//Search Startup values for enter the room
	fbSearchStartUpLevel 		: FB_SearchStartUpLevel_EX ;
	
END_VAR

VAR_IN_OUT
	stTuneData					: ST_TuneData_EX;
	stPirSensorData				: ST_DALI_Sensor;
	stLiveData					: ST_LiveData;
END_VAR

fbBallast(nCycleTimeInMS := nCycleTimeInMS);


A_TuningProcess();
A_RoomFct();

A_DaliUpdate();

ACTION A_DaliUpdate:

	IF stDaliSetup.DALI_LINE_NUM_PRIM <> 0 THEN
		
		stLgtCmd_Prim.bSetCtrlValDct:= fbLightCtrl_2Rows.bWriteValue ;
		stLgtCmd_Prim.fSetCtrlValDct:= fbLightCtrl_2Rows.fSP_Room;
		stLgtCmd_Prim.bDimDwn := fbLightCtrl_2Rows.bDimDwn;
		stLgtCmd_Prim.bDimUp := fbLightCtrl_2Rows.bDimUp;
		
		stLgtCmd_Prim.bClMinCtrlVal:= fbLightCtrl_2Rows.bClMinCtrlVal;
		
		fbBallast.M_PrimBallast(
				byShrtAdr_Prim:= stDaliSetup.byShrtAdr_Prim, 
				byGrpAdr_Prim:= stDaliSetup.byGrpAdr_Prim, 
				eMod_Prim:= stDaliSetup.eMod_Prim, 
				stLgtCmd_Prim:= stLgtCmd_Prim, 
				DALI_LINE_NUM:=stDaliSetup.DALI_LINE_NUM_PRIM,
				bUseGlobalFadeTimeSettings:= stDaliSetup.bLocal_GlobalFadeInfo , 
				bReInit:= bReInit, 
				bTurnOff:=fbLightCtrl.bOffZone1 , 
				ipCommunication:= ipCommunication_Prim );
	END_IF 
	
	IF stDaliSetup.DALI_LINE_NUM_SEC <> 0 THEN

		stLgtCmd_Sec.bSetCtrlValDct:= fbLightCtrl_2Rows.bWriteValue ;
		stLgtCmd_Sec.fSetCtrlValDct:=fbLightCtrl_2Rows.fSP_Window;
		stLgtCmd_Sec.bDimDwn := fbLightCtrl_2Rows.bDimDwn;
		stLgtCmd_Sec.bDimUp := fbLightCtrl_2Rows.bDimUp;		

		stLgtCmd_Sec.bClMinCtrlVal:= fbLightCtrl_2Rows.bClMinCtrlVal;
	
		fbBallast.M_SecBallast(
			byShrtAdr_Sec:= stDaliSetup.byShrtAdr_Sec, 
			byGrpAdr_Sec:= stDaliSetup.byGrpAdr_Sec, 
			eMod_Sec:= stDaliSetup.eMod_Sec, 
			stLgtCmd_Sec:= stLgtCmd_Sec, 
			DALI_LINE_NUM:=stDaliSetup.DALI_LINE_NUM_SEC,
			bUseGlobalFadeTimeSettings:= stDaliSetup.bLocal_GlobalFadeInfo , 
			bReInit:= bReInit, 
			bTurnOff:=fbLightCtrl.bOffZone2 , 
			ipCommunication:= ipCommunication_Sec );		
	END_IF 
	
	IF stDaliSetup.DALI_LINE_NUM_SUPL <> 0 THEN
	
		fbBallast.M_SuplBallast(
			byShrtAdr_Supl:= stDaliSetup.byShrtAdr_Supl, 
			byGrpAdr_Supl:= stDaliSetup.byGrpAdr_Supl, 
			eMod_Supl:= stDaliSetup.eMod_Supl, 
			stLgtCmd_Supl:= stLgtCmd_Supl, 
			DALI_LINE_NUM:=stDaliSetup.DALI_LINE_NUM_SUPL,
			bUseGlobalFadeTimeSettings:= stDaliSetup.bLocal_GlobalFadeInfo , 
			bReInit:= bReInit, 
			bTurnOff:= fbLightCtrl.bOffZone2 , 
			ipCommunication:= ipCommunication_Supl );
	END_IF
END_ACTION

ACTION A_RoomFct:

fbLightCtrl(
	bTopButtonZone1:= bButtonZone1,
	bBottomButtonZone1 := bBottomButtonZone1,
	bButtonZone2:= bButtonZone2,
	bTopButtonOverride:= bTopButtonOverride,
	bBottomButtonOverride:= bBottomButtonOverride,
	bNoButtons:= bNoButtons,
	bPIR:= stPirSensorData.bPrc, 
	fLuxOn:= fLuxOn, 
	fLuxDim:= fLuxDim, 
	tPIRDim:= tPIRDim, 
	tPIROff:= tPIROff, 
	fLuxZone1=> , 
	bDimUp=> , 
	bDimDwn=> , 
	bOnZone1=> bOccupiedRoom, 
	bOffZone1=> , 
	bAutoZone2=> , 
	bOnZone2=> , 
	bOffZone2=> );

bEnableLightCtrl:= fbLightCtrl.bOnZone1 AND fbLightCtrl.bAutoZone1;

fbRTrigStartCtrl(CLK:= fbAutoTuneStartUpLevels.bTuningDone AND bEnableLightCtrl);
fbStartStopLightCtrl(SET1 :=fbRTrigStartCtrl.Q , RESET:= NOT bEnableLightCtrl OR fbLightCtrl.bDimDwn OR fbLightCtrl.bDimUp );

fbSearchStartUpLevel(
	bSearch:= fbStartStopLightCtrl.Q1, 
	fSp:= fbLightCtrl.fLuxZone1, 
	stPirSensorData:= stPirSensorData, 
	bSync=> , 
	fSttUpCtrlVal=> , 
	stTuneData:=stTuneData );
	
fbLightCtrl_2Rows(
	_bEnable:=  fbStartStopLightCtrl.Q1, 
	_bSyncVal:=fbSearchStartUpLevel.bSync , 
	_fSyncVal:= fbSearchStartUpLevel.fSttUpCtrlVal, 
	_fSP:= fbLightCtrl.fLuxZone1, 
	_fPV:=stPirSensorData.fBrightness , 
	_fStep1Limit:= 8, 
	_fSPStep1:= 0.5, 
	_fStep2Limit:= 16, 
	_fSPStep2:= 1, 
	_fStep3Limit:= 24, 
	_fSPStep3:= 1.5, 
	_fStep4Limit:= 34, 
	_fSPStep4:= 2.0, 
	_fStep5Limit:= 40, 
	_fSPStep5:= 2.5, 
	_tStepTime:= T#10S, 																											//Testing 10s (originally 15s)
	_bStepModeCalculationOnSP:= FALSE , 
	_bTuningInProcess:= bTunningInProcess, 
	_bSetValDct:= fbAutoTuneStartUpLevels.bSetValDct, 
	_fSetValDct:= fbAutoTuneStartUpLevels.fSetValDct, 
	_bDimUp:= fbLightCtrl.bDimUp, 
	_bDimDown:= fbLightCtrl.bDimDwn, 
	_bOff:= fbLightCtrl.bOffZone1, 
	_fRowOffset:= fOffsetSec, 
	_fActlLgtLvl_Prim:= fbBallast.fActlLgtLvl_Prim, 
	_fActlLgtLvl_Sec:= fbBallast.fActlLgtLvl_Sec, 
	_bRecallManualLevel:= , 
	_fMinOutputPowerLevel := fMinOutputPowerLevelRoom ,
	_fMaxOutputPowerLevel := fMaxOutputPowerLevelRoom,
	_DALI_LINE_NUM_SEC	:= stDaliSetup.DALI_LINE_NUM_SEC,
	fSP_Window=> , 
	fSP_Room=> , 
	bWriteValue=> , 
	bDimUp=> , 
	bDimDwn=> , 
	bOff=> , 
	bClMinCtrlVal=> ,
	stPirSensorData:=stPirSensorData);
	
//Supplement light
fbLightCtrl_Supl(
	bSwi:= , 
	bSwiUp:= , 
	bSwiDwn:= , 
	udiSwiOvrTi:= , 
	bUp:= , 
	bDwn:= , 
	bOn:=fbLightCtrl.bOnZone2 , 
	bOff:= fbLightCtrl.bOffZone2, 
	eOnMod:= , 
	fOnVal:= , 
	bClMinVal:= , 
	bClMaxVal:= , 
	bSetValDct:= , 
	fSetValDct:= , 
	fActlLgtLvl:= fbBallast.fActlLgtLvl_Supl, 
	stLgtCmd=> stLgtCmd_Supl);
END_ACTION

ACTION A_TuningProcess:

fbAutoTuneStartUpLevels(
	bRunTuning:= (NOT stTuneData.bTunnigDone AND stPirSensorData.fBrightness < 25) OR bRunTuning, 
	tTuningDelay:= DALI_Param.tOutTuneDelay, 
	bTuningInProcess=> bTunningInProcess, 
	sActProcess=> , 
	bTuningDone=> , 
	bSetValDct=> , 
	fSetValDct=> , 
	stTuneData:=stTuneData,
 	stPirSensorData:= stPirSensorData);
END_ACTION

END_FUNCTION_BLOCK

// POUs/Templates/FB_Light_Type_B
FUNCTION_BLOCK FB_Light_Type_B
VAR_INPUT	
	nZoneID						: UDINT;
	bButtonZone1				: BOOL;
	bBottomButtonZone1			: BOOL;
	bButtonZone2				: BOOL;
	bTopButtonOverride		: BOOL;
	bBottomButtonOverride	: BOOL;
	bNoButtons					: BOOL;
	bNeighborRoomsPir			: BOOL;
	fLuxOn 						: REAL;
	fLuxDim						: REAL;
	tPIRDim						: TIME;
	tPIROff						: TIME;
	fOffsetSec					: REAL;
	bReInit						: BOOL;
	stDaliSetup					: ST_DALI_RoomSetup;
	ipCommunication_Prim		: I_DALICommunication;
	ipCommunication_Sec			: I_DALICommunication;
	ipCommunication_Supl		: I_DALICommunication;
	fMinOutputPowerLevelRoom 	: REAL;
	fMaxOutputPowerLevelRoom	: REAL;
	nCycleTimeInMS				: UDINT;
	bRunTuning 					: BOOL;
END_VAR
VAR_OUTPUT
	bOccupiedRoom 	: BOOL;
	bError_Prim 	: BOOL;
	nError_Prim 	: UINT;
END_VAR
VAR
	fbBallast					: FB_Light_Ballast;
	fbLightCtrl					: FB_FunctionType_A ;
	fbShortLongPresZone1 		: FB_Click;
	fbShortLongPressBottomZone1 : FB_Click;
	fbShortLongPresZone2 		: FB_Click;

	stLgtCmd_Prim				: ST_LgtCmd;
	stLgtCmd_Sec				: ST_LgtCmd;
	stLgtCmd_Supl				: ST_LgtCmd;
	
	fbLightCtrl_2Rows			: FB_LightCtrl_2Groups;
	fbLightCtrl_Supl			: FB_LightSwitch;

	bTunningInProcess			: BOOL;
	bEnableLightCtrl			: BOOL;
	fbRTrigStartCtrl 			: R_TRIG;
	
	bAnyPir						: BOOL;

//Tuning data
	fbPulsReadSensorData_TON	: TON;
	fbAutoTuneStartUpLevels		: FB_AutoTune_TcBA_Ex;
	fbR_TrigTuningDone			: R_TRIG ;
	fbStartStopLightCtrl: SR;
	
//Search Startup values for enter the room
	fbSearchStartUpLevel 		: FB_SearchStartUpLevel_EX ;
	
END_VAR

VAR_IN_OUT
	stTuneData					: ST_TuneData_EX;
	stPirSensorData				: ST_DALI_Sensor;
	stLiveData					: ST_LiveData;
END_VAR

fbBallast(nCycleTimeInMS := nCycleTimeInMS);


A_TuningProcess();
A_RoomFct();

A_DaliUpdate();

ACTION A_DaliUpdate:

	IF stDaliSetup.DALI_LINE_NUM_PRIM <> 0 THEN
		
		stLgtCmd_Prim.bSetCtrlValDct:= fbLightCtrl_2Rows.bWriteValue ;
		stLgtCmd_Prim.fSetCtrlValDct:= fbLightCtrl_2Rows.fSP_Room;
		stLgtCmd_Prim.bDimDwn := fbLightCtrl_2Rows.bDimDwn;
		stLgtCmd_Prim.bDimUp := fbLightCtrl_2Rows.bDimUp;
		
		stLgtCmd_Prim.bClMinCtrlVal:= fbLightCtrl_2Rows.bClMinCtrlVal;
		
		fbBallast.M_PrimBallast(
				byShrtAdr_Prim:= stDaliSetup.byShrtAdr_Prim, 
				byGrpAdr_Prim:= stDaliSetup.byGrpAdr_Prim, 
				eMod_Prim:= stDaliSetup.eMod_Prim, 
				stLgtCmd_Prim:= stLgtCmd_Prim, 
				DALI_LINE_NUM:=stDaliSetup.DALI_LINE_NUM_PRIM,
				bUseGlobalFadeTimeSettings:= stDaliSetup.bLocal_GlobalFadeInfo , 
				bReInit:= bReInit, 
				bTurnOff:=fbLightCtrl.bOffZone1 , 
				ipCommunication:= ipCommunication_Prim );
	END_IF 
	
	IF stDaliSetup.DALI_LINE_NUM_SEC <> 0 THEN

		stLgtCmd_Sec.bSetCtrlValDct:= fbLightCtrl_2Rows.bWriteValue ;
		stLgtCmd_Sec.fSetCtrlValDct:=fbLightCtrl_2Rows.fSP_Window;
		stLgtCmd_Sec.bDimDwn := fbLightCtrl_2Rows.bDimDwn;
		stLgtCmd_Sec.bDimUp := fbLightCtrl_2Rows.bDimUp;		

		stLgtCmd_Sec.bClMinCtrlVal:= fbLightCtrl_2Rows.bClMinCtrlVal;
	
		fbBallast.M_SecBallast(
			byShrtAdr_Sec:= stDaliSetup.byShrtAdr_Sec, 
			byGrpAdr_Sec:= stDaliSetup.byGrpAdr_Sec, 
			eMod_Sec:= stDaliSetup.eMod_Sec, 
			stLgtCmd_Sec:= stLgtCmd_Sec, 
			DALI_LINE_NUM:=stDaliSetup.DALI_LINE_NUM_SEC,
			bUseGlobalFadeTimeSettings:= stDaliSetup.bLocal_GlobalFadeInfo , 
			bReInit:= bReInit, 
			bTurnOff:=fbLightCtrl.bOffZone2 , 
			ipCommunication:= ipCommunication_Sec );		
	END_IF 
	
	IF stDaliSetup.DALI_LINE_NUM_SUPL <> 0 THEN
	
		fbBallast.M_SuplBallast(
			byShrtAdr_Supl:= stDaliSetup.byShrtAdr_Supl, 
			byGrpAdr_Supl:= stDaliSetup.byGrpAdr_Supl, 
			eMod_Supl:= stDaliSetup.eMod_Supl, 
			stLgtCmd_Supl:= stLgtCmd_Supl, 
			DALI_LINE_NUM:=stDaliSetup.DALI_LINE_NUM_SUPL,
			bUseGlobalFadeTimeSettings:= stDaliSetup.bLocal_GlobalFadeInfo , 
			bReInit:= bReInit, 
			bTurnOff:= fbLightCtrl.bOffZone2 , 
			ipCommunication:= ipCommunication_Supl );
	END_IF
END_ACTION

ACTION A_RoomFct:
bAnyPir	:= stPirSensorData.bPrc OR bNeighborRoomsPir;

fbLightCtrl(
	bTopButtonZone1:= bButtonZone1,
	bBottomButtonZone1 := bBottomButtonZone1,
	bButtonZone2:= bButtonZone2,
	bTopButtonOverride:= bTopButtonOverride,
	bBottomButtonOverride:= bBottomButtonOverride,
	bNoButtons:= bNoButtons,
	bPIR:= bAnyPir, 
	fLuxOn:= fLuxOn, 
	fLuxDim:= fLuxDim, 
	tPIRDim:= tPIRDim, 
	tPIROff:= tPIROff, 
	fLuxZone1=> , 
	bDimUp=> , 
	bDimDwn=> , 
	bOnZone1=> bOccupiedRoom, 
	bOffZone1=> , 
	bAutoZone2=> , 
	bOnZone2=> , 
	bOffZone2=> );

bEnableLightCtrl:= fbLightCtrl.bOnZone1 AND fbLightCtrl.bAutoZone1;

fbRTrigStartCtrl(CLK:= fbAutoTuneStartUpLevels.bTuningDone AND bEnableLightCtrl);
fbStartStopLightCtrl(SET1 :=fbRTrigStartCtrl.Q , RESET:= NOT bEnableLightCtrl OR fbLightCtrl.bDimDwn OR fbLightCtrl.bDimUp );

fbSearchStartUpLevel(
	bSearch:= fbStartStopLightCtrl.Q1, 
	fSp:= fbLightCtrl.fLuxZone1, 
	stPirSensorData:= stPirSensorData, 
	bSync=> , 
	fSttUpCtrlVal=> , 
	stTuneData:=stTuneData );
	
fbLightCtrl_2Rows(
	_bEnable:=  fbStartStopLightCtrl.Q1, 
	_bSyncVal:=fbSearchStartUpLevel.bSync , 
	_fSyncVal:= fbSearchStartUpLevel.fSttUpCtrlVal, 
	_fSP:= fbLightCtrl.fLuxZone1, 
	_fPV:=stPirSensorData.fBrightness , 
	_fStep1Limit:= 8, 
	_fSPStep1:= 0.5, 
	_fStep2Limit:= 16, 
	_fSPStep2:= 1, 
	_fStep3Limit:= 24, 
	_fSPStep3:= 1.5, 
	_fStep4Limit:= 34, 
	_fSPStep4:= 2.0, 
	_fStep5Limit:= 40, 
	_fSPStep5:= 2.5, 
	_tStepTime:= T#10S, 																											//Testing 10s (originally 15s)
	_bStepModeCalculationOnSP:= FALSE , 
	_bTuningInProcess:= bTunningInProcess, 
	_bSetValDct:= fbAutoTuneStartUpLevels.bSetValDct, 
	_fSetValDct:= fbAutoTuneStartUpLevels.fSetValDct, 
	_bDimUp:= fbLightCtrl.bDimUp, 
	_bDimDown:= fbLightCtrl.bDimDwn, 
	_bOff:= fbLightCtrl.bOffZone1, 
	_fRowOffset:= fOffsetSec, 
	_fActlLgtLvl_Prim:= fbBallast.fActlLgtLvl_Prim, 
	_fActlLgtLvl_Sec:= fbBallast.fActlLgtLvl_Sec, 
	_bRecallManualLevel:= , 
	_fMinOutputPowerLevel := fMinOutputPowerLevelRoom ,
	_fMaxOutputPowerLevel := fMaxOutputPowerLevelRoom,
	_DALI_LINE_NUM_SEC	:= stDaliSetup.DALI_LINE_NUM_SEC,
	fSP_Window=> , 
	fSP_Room=> , 
	bWriteValue=> , 
	bDimUp=> , 
	bDimDwn=> , 
	bOff=> , 
	bClMinCtrlVal=> ,
	stPirSensorData:=stPirSensorData);
	
//Supplement light
fbLightCtrl_Supl(
	bSwi:= , 
	bSwiUp:= , 
	bSwiDwn:= , 
	udiSwiOvrTi:= , 
	bUp:= , 
	bDwn:= , 
	bOn:=fbLightCtrl.bOnZone2 , 
	bOff:= fbLightCtrl.bOffZone2, 
	eOnMod:= , 
	fOnVal:= , 
	bClMinVal:= , 
	bClMaxVal:= , 
	bSetValDct:= , 
	fSetValDct:= , 
	fActlLgtLvl:= fbBallast.fActlLgtLvl_Supl, 
	stLgtCmd=> stLgtCmd_Supl);
END_ACTION

ACTION A_TuningProcess:

fbAutoTuneStartUpLevels(
	bRunTuning:= (NOT stTuneData.bTunnigDone AND stPirSensorData.fBrightness < 25) OR bRunTuning, 
	tTuningDelay:= DALI_Param.tOutTuneDelay, 
	bTuningInProcess=> bTunningInProcess, 
	sActProcess=> , 
	bTuningDone=> , 
	bSetValDct=> , 
	fSetValDct=> , 
	stTuneData:=stTuneData,
 	stPirSensorData:= stPirSensorData);
END_ACTION

END_FUNCTION_BLOCK

// Project Information/F_GetCompany
// This function has been automatically generated from the project information.
{attribute 'signature_flag' := '1073741824'}
{attribute 'TcGenerated'}
{attribute 'no-analysis'}
FUNCTION F_GetCompany : WSTRING
VAR_INPUT
	
END_VAR

F_GetCompany := "StroemHansen";

END_FUNCTION

// Project Information/F_GetTitle
// This function has been automatically generated from the project information.
{attribute 'signature_flag' := '1073741824'}
{attribute 'TcGenerated'}
{attribute 'no-analysis'}
FUNCTION F_GetTitle : WSTRING
VAR_INPUT
	
END_VAR

F_GetTitle := "SH_Light";

END_FUNCTION

// Project Information/F_GetVersion
// This function has been automatically generated from the project information.
{attribute 'signature_flag' := '1073741824'}
{attribute 'TcGenerated'}
{attribute 'no-analysis'}
FUNCTION F_GetVersion : ST_LibVersion
VAR_INPUT
	
END_VAR

F_GetVersion.iMajor := 3;
F_GetVersion.iMinor := 1;
F_GetVersion.iBuild := 5;
F_GetVersion.iRevision := 4;
F_GetVersion.sVersion := '3.1.5.4';
F_GetVersion.nFlags := 0;

END_FUNCTION
